// Mitsubishi GX Works2 project: Ex4   PLC: Q03UDV

PROGRAM MAIN
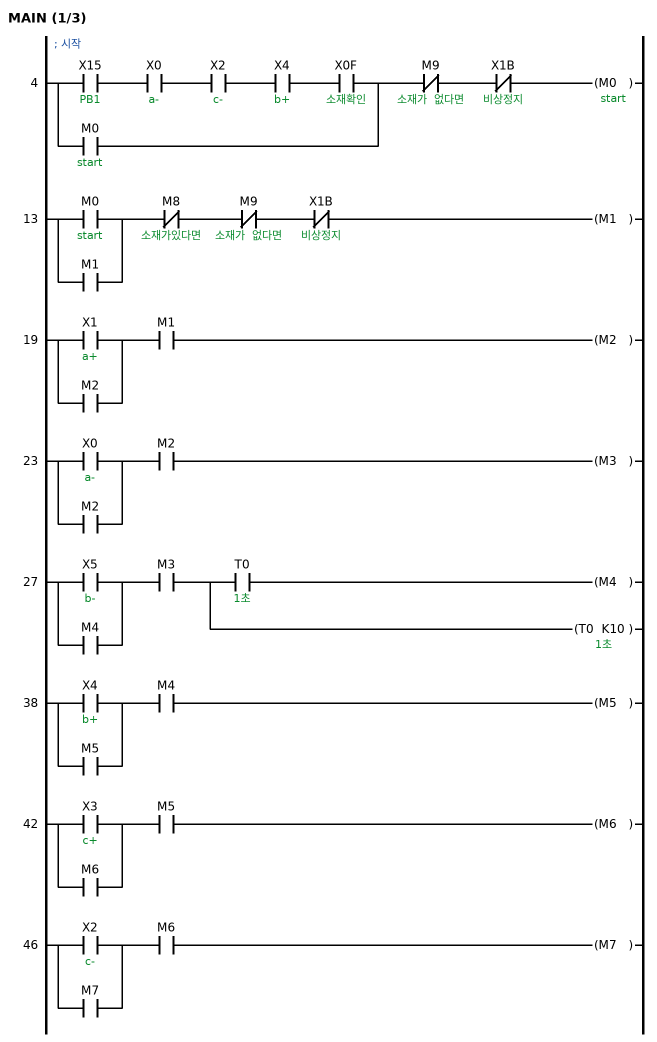
; 시작
4     LD      X15  ; PB1
      AND     X0  ; a-
      AND     X2  ; c-
      AND     X4  ; b+
      AND     X0F  ; 소재확인
      OR      M0  ; start
      ANI     M9  ; 소재가  없다면
      ANI     X1B  ; 비상정지
      OUT     M0  ; start
13    LD      M0  ; start
      OR      M1
      ANI     M8  ; 소재가있다면
      ANI     M9  ; 소재가  없다면
      ANI     X1B  ; 비상정지
      OUT     M1
19    LD      X1  ; a+
      OR      M2
      AND     M1
      OUT     M2
23    LD      X0  ; a-
      OR      M2
      AND     M2
      OUT     M3
27    LD      X5  ; b-
      OR      M4
      AND     M3
      MPS
      AND     T0  ; 1초
      OUT     M4
      MPP
      OUT     T0 K10  ; 1초
38    LD      X4  ; b+
      OR      M5
      AND     M4
      OUT     M5
42    LD      X3  ; c+
      OR      M6
      AND     M5
      OUT     M6
46    LD      X2  ; c-
      OR      M7
      AND     M6
      OUT     M7
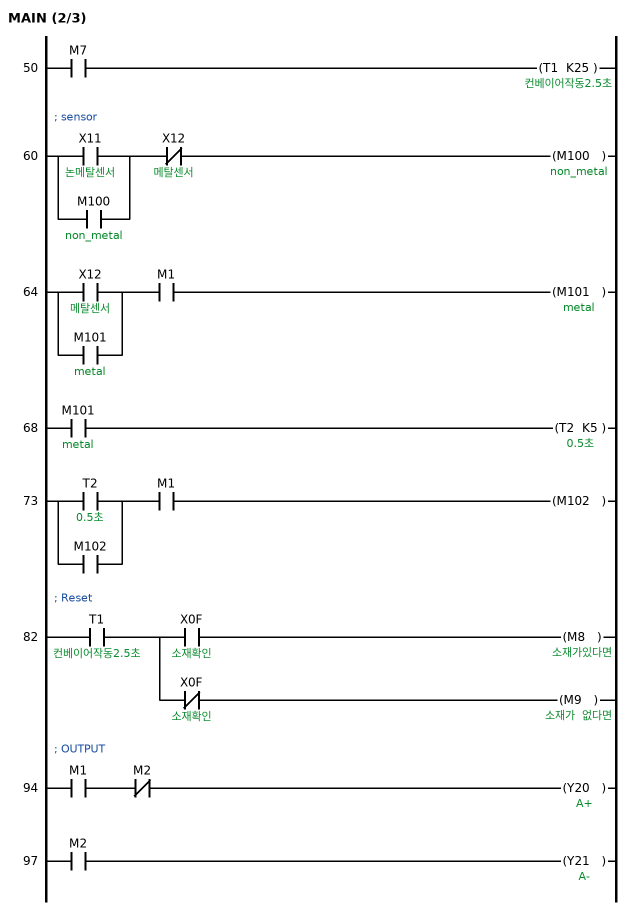
50    LD      M7
      OUT     T1 K25  ; 컨베이어작동2.5초
; sensor
60    LD      X11  ; 논메탈센서
      OR      M100  ; non_metal
      ANI     X12  ; 메탈센서
      OUT     M100  ; non_metal
64    LD      X12  ; 메탈센서
      OR      M101  ; metal
      AND     M1
      OUT     M101  ; metal
68    LD      M101  ; metal
      OUT     T2 K5  ; 0.5초
73    LD      T2  ; 0.5초
      OR      M102
      AND     M1
      OUT     M102
; Reset
82    LD      T1  ; 컨베이어작동2.5초
      MPS
      AND     X0F  ; 소재확인
      OUT     M8  ; 소재가있다면
      MPP
      ANI     X0F  ; 소재확인
      OUT     M9  ; 소재가  없다면
; OUTPUT
94    LD      M1
      ANI     M2
      OUT     Y20  ; A+
97    LD      M2
      OUT     Y21  ; A-
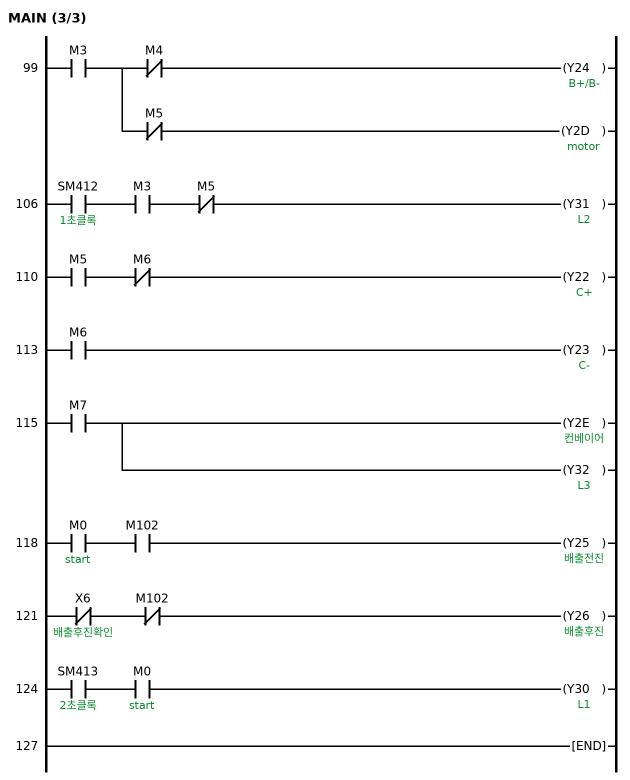
99    LD      M3
      MPS
      ANI     M4
      OUT     Y24  ; B+/B-
      MPP
      ANI     M5
      OUT     Y2D  ; motor
106   LD      SM412  ; 1초클록
      AND     M3
      ANI     M5
      OUT     Y31  ; L2
110   LD      M5
      ANI     M6
      OUT     Y22  ; C+
113   LD      M6
      OUT     Y23  ; C-
115   LD      M7
      OUT     Y2E  ; 컨베이어
      OUT     Y32  ; L3
118   LD      M0  ; start
      AND     M102
      OUT     Y25  ; 배출전진
121   LDI     X6  ; 배출후진확인
      ANI     M102
      OUT     Y26  ; 배출후진
124   LD      SM413  ; 2초클록
      AND     M0  ; start
      OUT     Y30  ; L1
127   END
END_PROGRAM
